// TIA Portal V20 export
// export: Created 2025-12-01T14:56:49.94347Z, ExportSetting None, DisplayName Totally Integrated Automation Portal, DisplayVersion V20 Update 3, DisplayName TIA Portal Openness, DisplayVersion V20 Update 3, DisplayName TIA Portal Version Control Interface, DisplayVersion V20 Update 3, DisplayName STEP 7 Professional, DisplayVersion V20 Update 3, DisplayName STEP 7 Safety, DisplayVersion V20 Update 2, DisplayName WinCC Basic/Comfort/Advanced, DisplayVersion V20 Update 3, DisplayName WinCC Professional, DisplayVersion V20 Update 3, DisplayName WinCC Unified, DisplayVersion V20 Update 3
FUNCTION_BLOCK "FB93_GALIBO_BarreraMedicion_P&F"   // FB93, LAD
{ S7_Optimized_Access := 'TRUE' }
// stored: AutoNumber false, MemoryReserve 100, SetENOAutomatically false
   VAR_INPUT
      Mesa : UInt;
      DIR_INI_Barrera : Int;
      NumGalibo : Int;
      Resolucion : Int;
      Offset : Int;
      Cota_Alt_Max : Int;
      pHs_Alt_Max : Bool;
      NodoOK_Barrera : Bool;
      PermisoLectura : Bool;
      Rearmar_ConMesaLibre : Bool;
   END_VAR
   VAR_OUTPUT
      Baliza : Bool;
      ErrorAltura : Bool;
      FinLectura : Bool;
   END_VAR
   VAR
      MemoriaAlturaBulto : Int;
      AlturaActual : Int;
      AlturaLeida_Puntos : Int;
      EstabilidadHaces : Int;
      BarreraSincronizada : Int;
      ObjetoBarrera : Int;
      AlturaBulto : Int;
   END_VAR
   VAR DB_SPECIFIC
      Altura_NOOK : Bool;
   END_VAR
   VAR
      G_ET00 : Bool;
      G_ET01 : Bool;
      G_ET02 : Bool;
   END_VAR
   VAR_TEMP
      NuevaAltura : Int;
      DatoValido : Bool;
      P_Barrera : DInt;
      EstadoZona : "EstadoZona";
      EstadoVI : "EstadosMesa";
   END_VAR
BEGIN

REGION Network 2: INICIALIZAR - Recoger las Variables de Estado de la Mesa
   // Se recoge - Estado_CBx
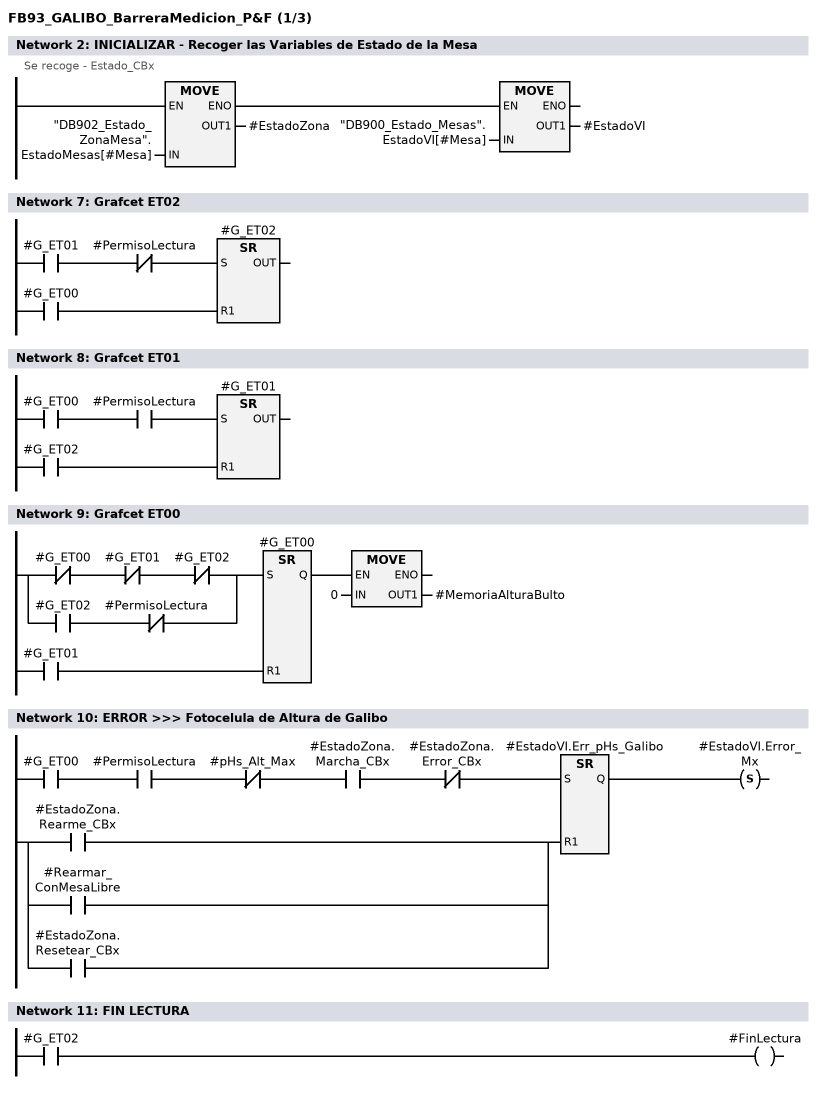
   RUNG wire#powerrail
      Move(in := "DB902_Estado_ZonaMesa".EstadoMesas[#Mesa], out1 => #EstadoZona)
      Move(in := "DB900_Estado_Mesas".EstadoVI[#Mesa], out1 => #EstadoVI)
   END_RUNG
   // the same network as SCL:
   #EstadoZona := "DB902_Estado_ZonaMesa".EstadoMesas[#Mesa];
   #EstadoVI := "DB900_Estado_Mesas".EstadoVI[#Mesa];
END_REGION

NETWORK
TITLE = INICIALIZAR
// -----------------------------------------------------------------------
// --- Inicializar

//////////////////////////////////////////////////////////////////////////////////
/// Leer las entradas de la Barrera

      L     0;  // Inicializo Variables
      T     #AlturaLeida_Puntos;



      AN    #NodoOK_Barrera;
      JC    _NoPresenteBarrera;  // Esta el nodo ?

      L     #DIR_INI_Barrera;  // Lectura del NBB - Numero de Beams Blocked
      SLD   3;
      T     #P_Barrera;

      L     IW [#P_Barrera];  // Dentro de Imagen
      L     W#16#1;  // cogemos el bit 0 y lo guardamos
      AW;
      T     #ObjetoBarrera;


      L     IW [#P_Barrera];  // Dentro de Imagen
      L     W#16#2;  // cogemos el bit 1 y lo guardamos
      AW;
      T     #BarreraSincronizada;

      L     IW [#P_Barrera];  // Dentro de Imagen
      L     W#16#4;  // cogemos el bit 2 y lo guardamos
      AW;
      T     #EstabilidadHaces;

      L     IW [#P_Barrera];
      SRD   4;  // eliminamos los primeros 4 bit, ya los hemos guardado anteriormente
      T     #AlturaLeida_Puntos;
////
//////      L     #NumberBeamsBlocked
//////      L     #Resolucion
//////      *I
//////      L     #Offset
//////      +I
//////      T     #AlturaTemporal
//////



NETWORK
TITLE = LEER ALTURA
// -----------------------------------------------------------------------
// --- Mirar si hay Lectura Nueva
      SET;
      A     #PermisoLectura;
      JC    LeerAltura;
//
//      L     0
//      T     #MemoriaAlturaBulto

      JU    FinFuncion;


LeerAltura:NOP   0;
      SET;
      L     #AlturaLeida_Puntos;
      L     0;
      <>I;
      =     #DatoValido;

      SET;
      AN    #DatoValido;
      JC    FinFuncion;



NETWORK
TITLE = Calcular Altura
// -----------------------------------------------------------------------
// --- Calcula la Altura Actual
// --- NuevaAltura = (LeidoAltura * Resolucion) + Offset

      L     #AlturaLeida_Puntos;
      L     #Resolucion;
      *I;
      L     #Offset;
      +I;
      T     #NuevaAltura;


// -----------------------------------------------------------------------
// --- Comprobar si es Mayor que la Nueva

      L     #NuevaAltura;  // Si la Altura Nueva
      L     #MemoriaAlturaBulto;  // Es Mayor o Igual
      >=I;
      JCN   FinFuncion;

      L     #NuevaAltura;  //////      L     #AlturaActual        // Guardo la Nueva Altura
      T     #MemoriaAlturaBulto;


NETWORK
TITLE = FINAL LECTURA
// --// -----------------------------------------------------------------------
// --- Se Acabo. Dar la Altura Memorizada

FinFuncion:NOP   0;

      L     #MemoriaAlturaBulto;  // Altura Maxima Leida
      T     #AlturaBulto;


//////
//////      L     #AlturaLeida_Puntos  // Altura Actual
//////      L     #Resolucion
//////      *I
//////      L     #Offset
//////      +I
//////      T     #AlturaActual
//////
      JU    fin;

_NoPresenteBarrera:NOP   0;
      L     0;
      T     #AlturaBulto;
fin:  NOP   0;



REGION Network 7: Grafcet ET02
   RUNG wire#powerrail
      Contact( #G_ET01 )
      I_Contact( #PermisoLectura )
      S_SR(operand := #G_ET02, r1 := wire#w1)
   END_RUNG
   RUNG wire#powerrail
      Contact( #G_ET00 )
   END_RUNG wire#w1
   // the same network as SCL:
   IF #G_ET01 AND NOT #PermisoLectura THEN
       #G_ET02 := TRUE;   // SR flip-flop
   END_IF;
   IF #G_ET00 THEN #G_ET02 := FALSE; END_IF;
END_REGION

REGION Network 8: Grafcet ET01
   RUNG wire#powerrail
      Contact( #G_ET00 )
      Contact( #PermisoLectura )
      S_SR(operand := #G_ET01, r1 := wire#w1)
   END_RUNG
   RUNG wire#powerrail
      Contact( #G_ET02 )
   END_RUNG wire#w1
   // the same network as SCL:
   IF #G_ET00 AND #PermisoLectura THEN
       #G_ET01 := TRUE;   // SR flip-flop
   END_IF;
   IF #G_ET02 THEN #G_ET01 := FALSE; END_IF;
END_REGION

REGION Network 9: Grafcet ET00
   RUNG wire#powerrail
      I_Contact( #G_ET00 )
      I_Contact( #G_ET01 )
      I_Contact( #G_ET02 )
      wire#w1
      S_SR(operand := #G_ET00, r1 := wire#w2)
      Move(in := 0, out1 => #MemoriaAlturaBulto)
   END_RUNG
   RUNG wire#powerrail
      Contact( #G_ET02 )
      I_Contact( #PermisoLectura )
   END_RUNG wire#w1
   RUNG wire#powerrail
      Contact( #G_ET01 )
   END_RUNG wire#w2
   // the same network as SCL:
   IF (NOT #G_ET00 AND NOT #G_ET01 AND NOT #G_ET02) OR (#G_ET02 AND NOT #PermisoLectura) THEN
       #G_ET00 := TRUE;   // SR flip-flop
   END_IF;
   IF #G_ET01 THEN #G_ET00 := FALSE; END_IF;
   IF #G_ET00 THEN #MemoriaAlturaBulto := 0; END_IF;
END_REGION

REGION Network 10: ERROR >>> Fotocelula de Altura de Galibo
   RUNG wire#powerrail
      Contact( #G_ET00 )
      Contact( #PermisoLectura )
      I_Contact( #pHs_Alt_Max )
      Contact( #EstadoZona.Marcha_CBx )
      I_Contact( #EstadoZona.Error_CBx )
      S_SR(operand := #EstadoVI.Err_pHs_Galibo, r1 := wire#w1)
      S_Coil( #EstadoVI.Error_Mx )
   END_RUNG
   RUNG wire#powerrail
      Contact( #EstadoZona.Rearme_CBx )
   END_RUNG wire#w1
   RUNG wire#powerrail
      Contact( #Rearmar_ConMesaLibre )
   END_RUNG wire#w1
   RUNG wire#powerrail
      Contact( #EstadoZona.Resetear_CBx )
   END_RUNG wire#w1
   // the same network as SCL:
   IF #G_ET00 AND #PermisoLectura AND NOT #pHs_Alt_Max AND #EstadoZona.Marcha_CBx AND NOT #EstadoZona.Error_CBx THEN
       #EstadoVI.Err_pHs_Galibo := TRUE;   // SR flip-flop
   END_IF;
   IF #EstadoZona.Rearme_CBx OR #Rearmar_ConMesaLibre OR #EstadoZona.Resetear_CBx THEN
       #EstadoVI.Err_pHs_Galibo := FALSE;
   END_IF;
   IF #EstadoVI.Err_pHs_Galibo THEN #EstadoVI.Error_Mx := TRUE; END_IF;
END_REGION

REGION Network 11: FIN LECTURA
   RUNG wire#powerrail
      Contact( #G_ET02 )
      Coil( #FinLectura )
   END_RUNG
   // the same network as SCL:
   #FinLectura := #G_ET02;
END_REGION

REGION Network 12: SALIDAS >>> RODILLOS - Codificacion del Galibo >>> Altura
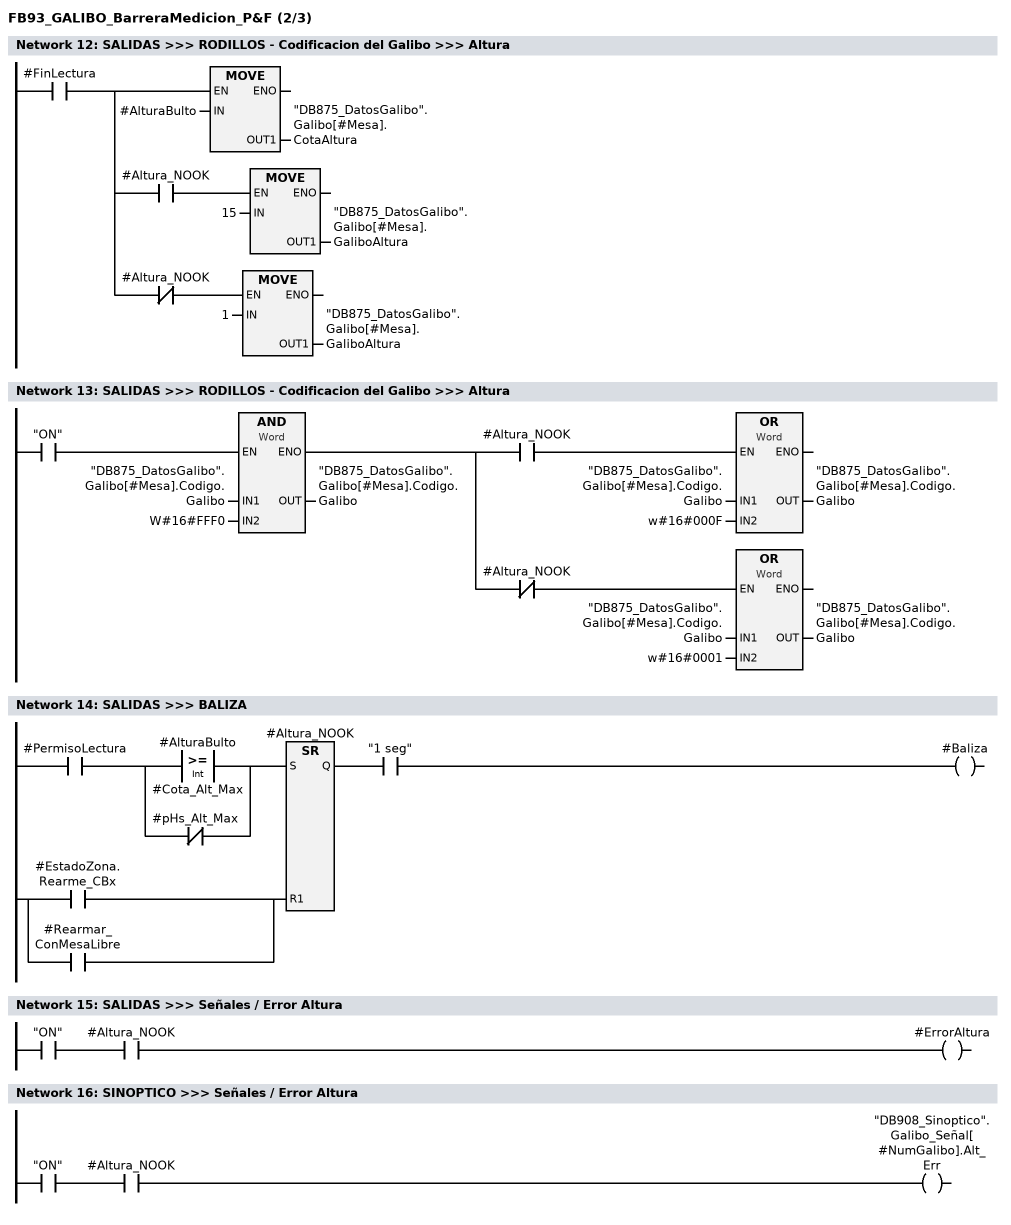
   RUNG wire#powerrail
      Contact( #FinLectura )
      wire#w1
      { S7_GenerateENO := "TRUE" } Move(in := #AlturaBulto, out1 => "DB875_DatosGalibo".Galibo[#Mesa].CotaAltura)
   END_RUNG
   RUNG wire#w1
      Contact( #Altura_NOOK )
      Move(in := 15, out1 => "DB875_DatosGalibo".Galibo[#Mesa].GaliboAltura)
   END_RUNG
   RUNG wire#w1
      I_Contact( #Altura_NOOK )
      Move(in := 1, out1 => "DB875_DatosGalibo".Galibo[#Mesa].GaliboAltura)
   END_RUNG
   // the same network as SCL:
   IF #FinLectura THEN "DB875_DatosGalibo".Galibo[#Mesa].CotaAltura := #AlturaBulto; END_IF;
   IF #FinLectura AND #Altura_NOOK THEN "DB875_DatosGalibo".Galibo[#Mesa].GaliboAltura := 15; END_IF;
   IF #FinLectura AND NOT #Altura_NOOK THEN "DB875_DatosGalibo".Galibo[#Mesa].GaliboAltura := 1; END_IF;
END_REGION

REGION Network 13: SALIDAS >>> RODILLOS - Codificacion del Galibo >>> Altura
   IF "ON" THEN
       "DB875_DatosGalibo".Galibo[#Mesa].Codigo.Galibo := "DB875_DatosGalibo".Galibo[#Mesa].Codigo.Galibo AND W#16#FFF0;
   END_IF;
   IF "ON" AND #Altura_NOOK THEN
       "DB875_DatosGalibo".Galibo[#Mesa].Codigo.Galibo := "DB875_DatosGalibo".Galibo[#Mesa].Codigo.Galibo OR w#16#000F;
   END_IF;
   IF "ON" AND NOT #Altura_NOOK THEN
       "DB875_DatosGalibo".Galibo[#Mesa].Codigo.Galibo := "DB875_DatosGalibo".Galibo[#Mesa].Codigo.Galibo OR w#16#0001;
   END_IF;
END_REGION

REGION Network 14: SALIDAS >>> BALIZA
   RUNG wire#powerrail
      Contact( #PermisoLectura )
      wire#w1
      { S7_Templates := "SrcType := Int" } GE_Contact(in1 := #AlturaBulto, in2 := #Cota_Alt_Max)
      wire#w2
      S_SR(operand := #Altura_NOOK, r1 := wire#w3)
      Contact( "1 seg" )
      Coil( #Baliza )
   END_RUNG
   RUNG wire#w1
      I_Contact( #pHs_Alt_Max )
   END_RUNG wire#w2
   RUNG wire#powerrail
      Contact( #EstadoZona.Rearme_CBx )
   END_RUNG wire#w3
   RUNG wire#powerrail
      Contact( #Rearmar_ConMesaLibre )
   END_RUNG wire#w3
   // the same network as SCL:
   IF #PermisoLectura AND ((#AlturaBulto >= #Cota_Alt_Max) OR NOT #pHs_Alt_Max) THEN
       #Altura_NOOK := TRUE;   // SR flip-flop
   END_IF;
   IF #EstadoZona.Rearme_CBx OR #Rearmar_ConMesaLibre THEN #Altura_NOOK := FALSE; END_IF;
   #Baliza := #Altura_NOOK AND "1 seg";
END_REGION

REGION Network 15: SALIDAS >>> Señales / Error Altura
   RUNG wire#powerrail
      Contact( "ON" )
      Contact( #Altura_NOOK )
      Coil( #ErrorAltura )
   END_RUNG
   // the same network as SCL:
   #ErrorAltura := "ON" AND #Altura_NOOK;
END_REGION

REGION Network 16: SINOPTICO >>> Señales / Error Altura
   RUNG wire#powerrail
      Contact( "ON" )
      Contact( #Altura_NOOK )
      Coil( "DB908_Sinoptico".Galibo_Señal[#NumGalibo].Alt_Err )
   END_RUNG
   // the same network as SCL:
   "DB908_Sinoptico".Galibo_Señal[#NumGalibo].Alt_Err := "ON" AND #Altura_NOOK;
END_REGION

REGION Network 17: SINOPTICO >>> Codigo
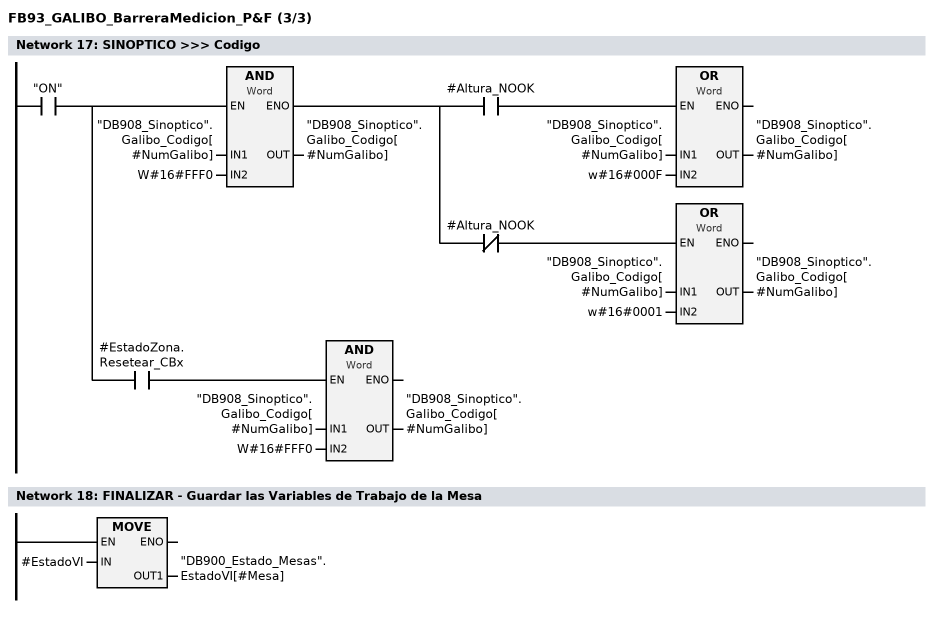
   IF "ON" THEN
       "DB908_Sinoptico".Galibo_Codigo[#NumGalibo] := "DB908_Sinoptico".Galibo_Codigo[#NumGalibo] AND W#16#FFF0;
   END_IF;
   IF "ON" AND #Altura_NOOK THEN
       "DB908_Sinoptico".Galibo_Codigo[#NumGalibo] := "DB908_Sinoptico".Galibo_Codigo[#NumGalibo] OR w#16#000F;
   END_IF;
   IF "ON" AND NOT #Altura_NOOK THEN
       "DB908_Sinoptico".Galibo_Codigo[#NumGalibo] := "DB908_Sinoptico".Galibo_Codigo[#NumGalibo] OR w#16#0001;
   END_IF;
   IF "ON" AND #EstadoZona.Resetear_CBx THEN
       "DB908_Sinoptico".Galibo_Codigo[#NumGalibo] := "DB908_Sinoptico".Galibo_Codigo[#NumGalibo] AND W#16#FFF0;
   END_IF;
END_REGION

REGION Network 18: FINALIZAR - Guardar las Variables de Trabajo de la Mesa
   RUNG wire#powerrail
      Move(in := #EstadoVI, out1 => "DB900_Estado_Mesas".EstadoVI[#Mesa])
   END_RUNG
   // the same network as SCL:
   "DB900_Estado_Mesas".EstadoVI[#Mesa] := #EstadoVI;
END_REGION
END_FUNCTION_BLOCK
